(* PLC project Tc3_EventLogger.Subscribe Demo, tc3-libraries-kb TwinCAT 3.1 *)
(* stored: creationDateTime 2026-05-11T01:00:00, modificationDateTime 2026-05-11T01:00:00 *)

PROGRAM P_Demo_Subscribe
  VAR
    fbListener : FB_ListenerBase2;  (* listener 实例 *)
    bSubscribed : BOOL;  (* 订阅 latch *)
    hr : HRESULT;  (* 返回值监视 *)
  END_VAR

// =============================================================================
// 场景：订阅所有 alarm + message 事件
// 价值：一次调用完成订阅，后续周期 Execute 即可收事件
// 验证：登录后 monitor bSubscribed 第一周期变 TRUE
// 验证步骤：
//   1. 右键 PLC 项目 → Import PLCopenXML → 选本文件
//   2. 引用 Tc3_EventLogger（System → References → Add library）
//   3. 编译 → 登录 → 运行；按 verify 注释里给出的在线写值操作
// =============================================================================

IF NOT bSubscribed THEN
    hr := fbListener.Subscribe(
        ipMessageFilterConfig := 0,            // 接收全部 message
        ipAlarmFilterConfig := 0);             // 接收全部 alarm
    bSubscribed := SUCCEEDED(hr);
END_IF;
END_PROGRAM
